TYPE "PositioningMachine_DataOut"
VERSION : 0.1
// Block: PositioningMachine_DataOut
   STRUCT
      Fan_M_Contactor : Bool;
   END_STRUCT;

END_TYPE
